// TIA Portal V20 export
FUNCTION_BLOCK "CentralShifter_SideShifters"   // FB17, LAD
{ S7_Optimized_Access := 'TRUE' }
// stored: MemoryReserve 100, SetENOAutomatically false
   VAR_INPUT
      In_Side_Drive_Pos : Bool;
      Position_CS : Int;
   END_VAR
   VAR_OUTPUT
      qLeftSide_in_Mid : Bool;
      qRightSide_in_Mid : Bool;
   END_VAR
   VAR
      Side_Hydraulic_CS_RL { S7_SetPoint := 'True'} : "Side_Hydraulic";
      Side_Hydraulic_CS_RR { S7_SetPoint := 'True'} : "Side_Hydraulic";
      Side_Driver_CS { S7_SetPoint := 'True'} : "Side_Driver";
      RL_Speed { S7_SetPoint := 'True'} : Int;
      RP_Speed : Int;
      CentralShifter_Side_Auto_Instance { S7_SetPoint := 'True'} : "CentralShifter_Side_Auto";
      SL_Auto_Speed { S7_SetPoint := 'True'} : Int;
      SR_Auto_Speed : Int;
      SL_Auto_Forward : Bool;
      SL_Auto_Backward : Bool;
      SR_Auto_Forward : Bool;
      SR_Auto_Backward : Bool;
      Sides_In_Position : Bool;
      Sides_In_H3_Pos : Bool;
      Sides_In_H5_Pos : Bool;
      Sides_In_CS_Pos : Bool;
      LightUp : Bool;
      LightMid : Bool;
      LightDown : Bool;
      SR_Error_Laser : Bool;
      SL_Error_Laser : Bool;
      Auto_Position_RL_Up : DInt;
      Auto_Position_RL_Mid : DInt;
      Auto_Position_RL_Down : DInt;
      Auto_Position_RR_Up : DInt;
      Auto_Position_RR_Mid : DInt;
      Auto_Position_RR_Down : DInt;
      Auto_Correction_RR : Int;
   END_VAR
   VAR RETAIN
      Stations : Array[7..13] of "CS_Sides_Stations";
   END_VAR
   VAR
      Status_Side_Go_H3 { S7_SetPoint := 'True'} : Int;
      Status_Side_Go_H5 : Int;
      Status_Side_Go_CS : Int;
      Auto_Hydraulic_Permission_H3 : Bool;
      Auto_Hydraulic_Permission_H5 : Bool;
      Auto_Hydraulic_Up_Timer { S7_SetPoint := 'True'} : TP_TIME;
      Auto_Hydraulic_Down_Timer { S7_SetPoint := 'True'} : TP_TIME;
      Station_H3_Empty : Bool;
      Station_H5_Empty : Bool;
      CS_R1_Sen_Up : Bool;
      CS_R1_Sen_Down : Bool;
      CS_R2_Sen_Up : Bool;
      CS_R2_Sen_Down : Bool;
      Auto_hyd_Up : Bool;
      Auto_hyd_Down : Bool;
      Hyd_Up_Status : Int;
      Hyd_Down_Status : Int;
      CS_RL_Error_Hyd : Bool;
      CS_RR_Error_Hyd : Bool;
      CS_Error_Hyd : Bool;
      CS_Error_Drive : Bool;
   END_VAR
   VAR CONSTANT
      Tolerance : Int := 60;
   END_VAR
   // Stations[7].RL_H3_Pos := 13516;
   // Stations[8].RL_H3_Pos := 13505;
   // Stations[9].RL_H3_Pos := 13520;
   // Stations[10].RL_H3_Pos := 13522;
   // Stations[11].RL_H3_Pos := 13526;
   // Stations[12].RL_H3_Pos := 13505;
   // Stations[13].RL_H3_Pos := 13500;
   // Stations[7].RR_H3_Pos := 13523;
   // Stations[8].RR_H3_Pos := 13495;
   // Stations[9].RR_H3_Pos := 13518;
   // Stations[10].RR_H3_Pos := 13527;
   // Stations[11].RR_H3_Pos := 13524;
   // Stations[12..13].RR_H3_Pos := 13525;
   // Stations[7].RL_Mid_Pos := 7915;
   // Stations[8].RL_Mid_Pos := 7910;
   // Stations[9].RL_Mid_Pos := 7933;
   // Stations[10].RL_Mid_Pos := 7928;
   // Stations[11].RL_Mid_Pos := 7937;
   // Stations[12].RL_Mid_Pos := 7932;
   // Stations[13].RL_Mid_Pos := 7916;
   // Stations[7].RR_Mid_Pos := 7925;
   // Stations[8].RR_Mid_Pos := 7895;
   // Stations[9].RR_Mid_Pos := 7922;
   // Stations[10].RR_Mid_Pos := 7935;
   // Stations[11].RR_Mid_Pos := 7926;
   // Stations[12].RR_Mid_Pos := 7932;
   // Stations[13].RR_Mid_Pos := 7939;
   // Stations[7].RL_H5_Pos := 1930;
   // Stations[8].RL_H5_Pos := 1917;
   // Stations[9].RL_H5_Pos := 1928;
   // Stations[10].RL_H5_Pos := 1929;
   // Stations[11].RL_H5_Pos := 1936;
   // Stations[12].RL_H5_Pos := 1924;
   // Stations[13].RL_H5_Pos := 1918;
   // Stations[7].RR_H5_Pos := 1929;
   // Stations[8].RR_H5_Pos := 1900;
   // Stations[9].RR_H5_Pos := 1921;
   // Stations[10].RR_H5_Pos := 1933;
   // Stations[11].RR_H5_Pos := 1928;
   // Stations[12].RR_H5_Pos := 1934;
   // Stations[13].RR_H5_Pos := 1915;
   // Stations[7].Correction := -20;
   // Stations[8].Correction := -15;
   // Stations[9].Correction := -5;
   // Stations[11].Correction := 0;
   // Stations[12].Correction := 10;
   // Stations[13].Correction := 15;
BEGIN

REGION Network 1: Hydraulic_RL
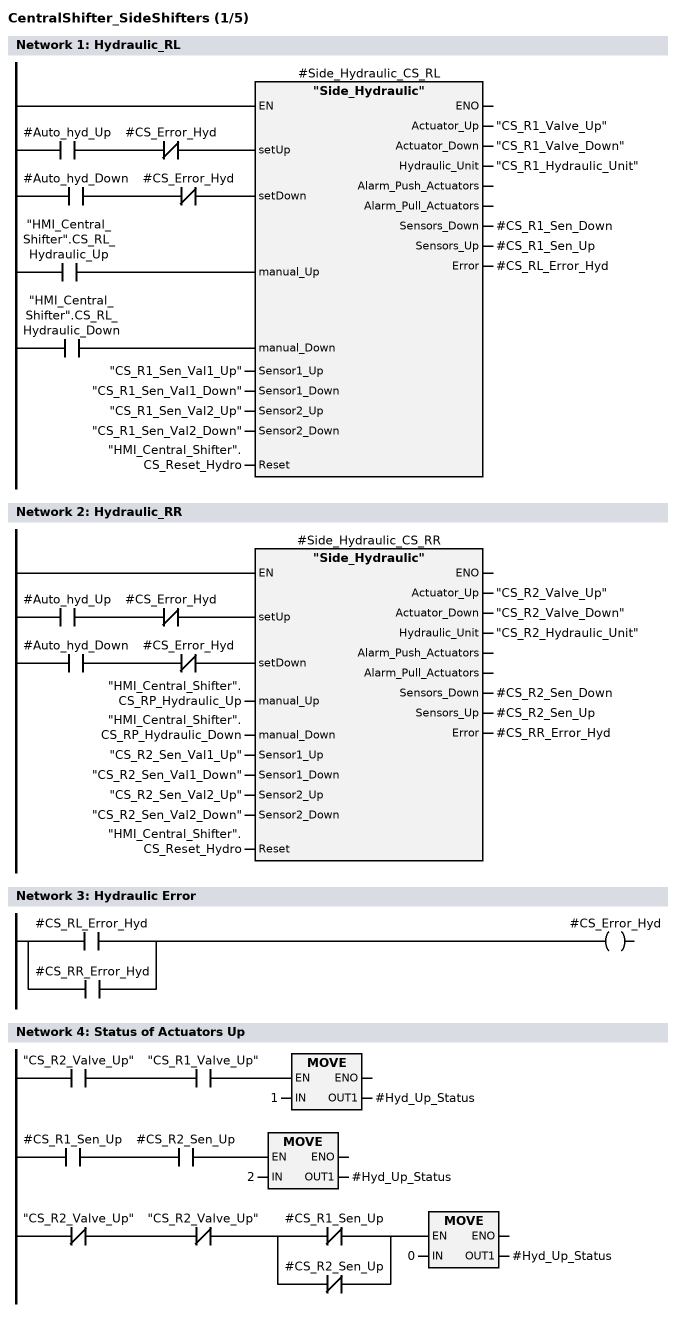
   RUNG wire#powerrail
      #Side_Hydraulic_CS_RL(setUp := wire#w1, setDown := wire#w2, manual_Up := wire#w3, manual_Down := wire#w4, Sensor1_Up := "CS_R1_Sen_Val1_Up", Sensor1_Down := "CS_R1_Sen_Val1_Down", Sensor2_Up := "CS_R1_Sen_Val2_Up", Sensor2_Down := "CS_R1_Sen_Val2_Down", Reset := "HMI_Central_Shifter".CS_Reset_Hydro, Actuator_Up => "CS_R1_Valve_Up", Actuator_Down => "CS_R1_Valve_Down", Hydraulic_Unit => "CS_R1_Hydraulic_Unit", Alarm_Push_Actuators =>, Alarm_Pull_Actuators =>, Sensors_Down => #CS_R1_Sen_Down, Sensors_Up => #CS_R1_Sen_Up, Error => #CS_RL_Error_Hyd)
   END_RUNG
   RUNG wire#powerrail
      Contact( #Auto_hyd_Up )
      I_Contact( #CS_Error_Hyd )
   END_RUNG wire#w1
   RUNG wire#powerrail
      Contact( #Auto_hyd_Down )
      I_Contact( #CS_Error_Hyd )
   END_RUNG wire#w2
   RUNG wire#powerrail
      Contact( "HMI_Central_Shifter".CS_RL_Hydraulic_Up )
   END_RUNG wire#w3
   RUNG wire#powerrail
      Contact( "HMI_Central_Shifter".CS_RL_Hydraulic_Down )
   END_RUNG wire#w4
   // the same network as SCL:
   #Side_Hydraulic_CS_RL(setUp := #Auto_hyd_Up AND NOT #CS_Error_Hyd,   // "Side_Hydraulic"
                         setDown := #Auto_hyd_Down AND NOT #CS_Error_Hyd,
                         manual_Up := "HMI_Central_Shifter".CS_RL_Hydraulic_Up,
                         manual_Down := "HMI_Central_Shifter".CS_RL_Hydraulic_Down,
                         Sensor1_Up := "CS_R1_Sen_Val1_Up",
                         Sensor1_Down := "CS_R1_Sen_Val1_Down",
                         Sensor2_Up := "CS_R1_Sen_Val2_Up",
                         Sensor2_Down := "CS_R1_Sen_Val2_Down",
                         Reset := "HMI_Central_Shifter".CS_Reset_Hydro,
                         Actuator_Up => "CS_R1_Valve_Up",
                         Actuator_Down => "CS_R1_Valve_Down",
                         Hydraulic_Unit => "CS_R1_Hydraulic_Unit",
                         Sensors_Down => #CS_R1_Sen_Down,
                         Sensors_Up => #CS_R1_Sen_Up,
                         Error => #CS_RL_Error_Hyd);
END_REGION

REGION Network 2: Hydraulic_RR
   RUNG wire#powerrail
      #Side_Hydraulic_CS_RR(setUp := wire#w1, setDown := wire#w2, manual_Up := "HMI_Central_Shifter".CS_RP_Hydraulic_Up, manual_Down := "HMI_Central_Shifter".CS_RP_Hydraulic_Down, Sensor1_Up := "CS_R2_Sen_Val1_Up", Sensor1_Down := "CS_R2_Sen_Val1_Down", Sensor2_Up := "CS_R2_Sen_Val2_Up", Sensor2_Down := "CS_R2_Sen_Val2_Down", Reset := "HMI_Central_Shifter".CS_Reset_Hydro, Actuator_Up => "CS_R2_Valve_Up", Actuator_Down => "CS_R2_Valve_Down", Hydraulic_Unit => "CS_R2_Hydraulic_Unit", Alarm_Push_Actuators =>, Alarm_Pull_Actuators =>, Sensors_Down => #CS_R2_Sen_Down, Sensors_Up => #CS_R2_Sen_Up, Error => #CS_RR_Error_Hyd)
   END_RUNG
   RUNG wire#powerrail
      Contact( #Auto_hyd_Up )
      I_Contact( #CS_Error_Hyd )
   END_RUNG wire#w1
   RUNG wire#powerrail
      Contact( #Auto_hyd_Down )
      I_Contact( #CS_Error_Hyd )
   END_RUNG wire#w2
   // the same network as SCL:
   #Side_Hydraulic_CS_RR(setUp := #Auto_hyd_Up AND NOT #CS_Error_Hyd,   // "Side_Hydraulic"
                         setDown := #Auto_hyd_Down AND NOT #CS_Error_Hyd,
                         manual_Up := "HMI_Central_Shifter".CS_RP_Hydraulic_Up,
                         manual_Down := "HMI_Central_Shifter".CS_RP_Hydraulic_Down,
                         Sensor1_Up := "CS_R2_Sen_Val1_Up",
                         Sensor1_Down := "CS_R2_Sen_Val1_Down",
                         Sensor2_Up := "CS_R2_Sen_Val2_Up",
                         Sensor2_Down := "CS_R2_Sen_Val2_Down",
                         Reset := "HMI_Central_Shifter".CS_Reset_Hydro,
                         Actuator_Up => "CS_R2_Valve_Up",
                         Actuator_Down => "CS_R2_Valve_Down",
                         Hydraulic_Unit => "CS_R2_Hydraulic_Unit",
                         Sensors_Down => #CS_R2_Sen_Down,
                         Sensors_Up => #CS_R2_Sen_Up,
                         Error => #CS_RR_Error_Hyd);
END_REGION

REGION Network 3: Hydraulic Error
   RUNG wire#powerrail
      Contact( #CS_RL_Error_Hyd )
      wire#w1
      Coil( #CS_Error_Hyd )
   END_RUNG
   RUNG wire#powerrail
      Contact( #CS_RR_Error_Hyd )
   END_RUNG wire#w1
   // the same network as SCL:
   #CS_Error_Hyd := #CS_RL_Error_Hyd OR #CS_RR_Error_Hyd;
END_REGION

REGION Network 4: Status of Actuators Up
   RUNG wire#powerrail
      Contact( "CS_R2_Valve_Up" )
      Contact( "CS_R1_Valve_Up" )
      Move(in := 1, out1 => #Hyd_Up_Status)
   END_RUNG
   RUNG wire#powerrail
      Contact( #CS_R1_Sen_Up )
      Contact( #CS_R2_Sen_Up )
      Move(in := 2, out1 => #Hyd_Up_Status)
   END_RUNG
   RUNG wire#powerrail
      I_Contact( "CS_R2_Valve_Up" )
      I_Contact( "CS_R2_Valve_Up" )
      wire#w1
      I_Contact( #CS_R1_Sen_Up )
      wire#w2
      Move(in := 0, out1 => #Hyd_Up_Status)
   END_RUNG
   RUNG wire#w1
      I_Contact( #CS_R2_Sen_Up )
   END_RUNG wire#w2
   // the same network as SCL:
   IF "CS_R2_Valve_Up" AND "CS_R1_Valve_Up" THEN #Hyd_Up_Status := 1; END_IF;
   IF #CS_R1_Sen_Up AND #CS_R2_Sen_Up THEN #Hyd_Up_Status := 2; END_IF;
   IF NOT "CS_R2_Valve_Up" AND NOT "CS_R2_Valve_Up" AND (NOT #CS_R1_Sen_Up OR NOT #CS_R2_Sen_Up) THEN
       #Hyd_Up_Status := 0;
   END_IF;
END_REGION

REGION Network 5: Status of Actuators Down
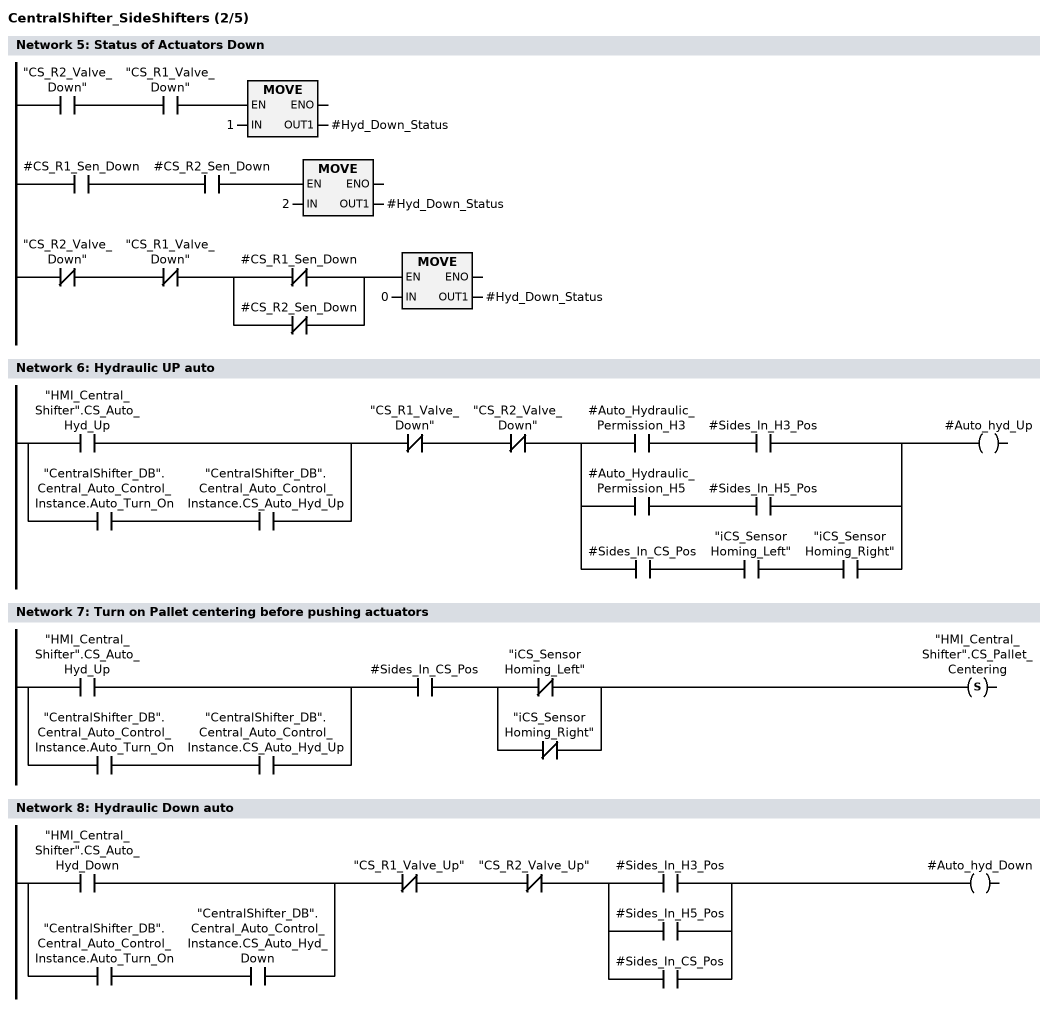
   RUNG wire#powerrail
      Contact( "CS_R2_Valve_Down" )
      Contact( "CS_R1_Valve_Down" )
      Move(in := 1, out1 => #Hyd_Down_Status)
   END_RUNG
   RUNG wire#powerrail
      Contact( #CS_R1_Sen_Down )
      Contact( #CS_R2_Sen_Down )
      Move(in := 2, out1 => #Hyd_Down_Status)
   END_RUNG
   RUNG wire#powerrail
      I_Contact( "CS_R2_Valve_Down" )
      I_Contact( "CS_R1_Valve_Down" )
      wire#w1
      I_Contact( #CS_R1_Sen_Down )
      wire#w2
      Move(in := 0, out1 => #Hyd_Down_Status)
   END_RUNG
   RUNG wire#w1
      I_Contact( #CS_R2_Sen_Down )
   END_RUNG wire#w2
   // the same network as SCL:
   IF "CS_R2_Valve_Down" AND "CS_R1_Valve_Down" THEN #Hyd_Down_Status := 1; END_IF;
   IF #CS_R1_Sen_Down AND #CS_R2_Sen_Down THEN #Hyd_Down_Status := 2; END_IF;
   IF NOT "CS_R2_Valve_Down" AND NOT "CS_R1_Valve_Down" AND (NOT #CS_R1_Sen_Down OR NOT #CS_R2_Sen_Down) THEN
       #Hyd_Down_Status := 0;
   END_IF;
END_REGION

REGION Network 6: Hydraulic UP auto
   RUNG wire#powerrail
      Contact( "HMI_Central_Shifter".CS_Auto_Hyd_Up )
      wire#w1
      I_Contact( "CS_R1_Valve_Down" )
      I_Contact( "CS_R2_Valve_Down" )
      wire#w2
      Contact( #Auto_Hydraulic_Permission_H3 )
      Contact( #Sides_In_H3_Pos )
      wire#w3
      Coil( #Auto_hyd_Up )
   END_RUNG
   RUNG wire#powerrail
      Contact( "CentralShifter_DB".Central_Auto_Control_Instance.Auto_Turn_On )
      Contact( "CentralShifter_DB".Central_Auto_Control_Instance.CS_Auto_Hyd_Up )
   END_RUNG wire#w1
   RUNG wire#w2
      Contact( #Auto_Hydraulic_Permission_H5 )
      Contact( #Sides_In_H5_Pos )
   END_RUNG wire#w3
   RUNG wire#w2
      Contact( #Sides_In_CS_Pos )
      Contact( "iCS_SensorHoming_Left" )
      Contact( "iCS_SensorHoming_Right" )
   END_RUNG wire#w3
   // the same network as SCL:
   #Auto_hyd_Up := ("HMI_Central_Shifter".CS_Auto_Hyd_Up OR ("CentralShifter_DB".Central_Auto_Control_Instance.Auto_Turn_On AND "CentralShifter_DB".Central_Auto_Control_Instance.CS_Auto_Hyd_Up)) AND NOT "CS_R1_Valve_Down" AND NOT "CS_R2_Valve_Down" AND ((#Auto_Hydraulic_Permission_H3 AND #Sides_In_H3_Pos) OR (#Auto_Hydraulic_Permission_H5 AND #Sides_In_H5_Pos) OR (#Sides_In_CS_Pos AND "iCS_SensorHoming_Left" AND "iCS_SensorHoming_Right"));
END_REGION

REGION Network 7: Turn on Pallet centering before pushing actuators
   RUNG wire#powerrail
      Contact( "HMI_Central_Shifter".CS_Auto_Hyd_Up )
      wire#w1
      Contact( #Sides_In_CS_Pos )
      wire#w2
      I_Contact( "iCS_SensorHoming_Left" )
      wire#w3
      S_Coil( "HMI_Central_Shifter".CS_Pallet_Centering )
   END_RUNG
   RUNG wire#powerrail
      Contact( "CentralShifter_DB".Central_Auto_Control_Instance.Auto_Turn_On )
      Contact( "CentralShifter_DB".Central_Auto_Control_Instance.CS_Auto_Hyd_Up )
   END_RUNG wire#w1
   RUNG wire#w2
      I_Contact( "iCS_SensorHoming_Right" )
   END_RUNG wire#w3
   // the same network as SCL:
   IF ("HMI_Central_Shifter".CS_Auto_Hyd_Up OR ("CentralShifter_DB".Central_Auto_Control_Instance.Auto_Turn_On AND "CentralShifter_DB".Central_Auto_Control_Instance.CS_Auto_Hyd_Up)) AND #Sides_In_CS_Pos AND (NOT "iCS_SensorHoming_Left" OR NOT "iCS_SensorHoming_Right") THEN
       "HMI_Central_Shifter".CS_Pallet_Centering := TRUE;
   END_IF;
END_REGION

REGION Network 8: Hydraulic Down auto
   RUNG wire#powerrail
      Contact( "HMI_Central_Shifter".CS_Auto_Hyd_Down )
      wire#w1
      I_Contact( "CS_R1_Valve_Up" )
      I_Contact( "CS_R2_Valve_Up" )
      wire#w2
      Contact( #Sides_In_H3_Pos )
      wire#w3
      Coil( #Auto_hyd_Down )
   END_RUNG
   RUNG wire#powerrail
      Contact( "CentralShifter_DB".Central_Auto_Control_Instance.Auto_Turn_On )
      Contact( "CentralShifter_DB".Central_Auto_Control_Instance.CS_Auto_Hyd_Down )
   END_RUNG wire#w1
   RUNG wire#w2
      Contact( #Sides_In_H5_Pos )
   END_RUNG wire#w3
   RUNG wire#w2
      Contact( #Sides_In_CS_Pos )
   END_RUNG wire#w3
   // the same network as SCL:
   #Auto_hyd_Down := ("HMI_Central_Shifter".CS_Auto_Hyd_Down OR ("CentralShifter_DB".Central_Auto_Control_Instance.Auto_Turn_On AND "CentralShifter_DB".Central_Auto_Control_Instance.CS_Auto_Hyd_Down)) AND NOT "CS_R1_Valve_Up" AND NOT "CS_R2_Valve_Up" AND (#Sides_In_H3_Pos OR #Sides_In_H5_Pos OR #Sides_In_CS_Pos);
END_REGION

REGION Network 9: Laser Error
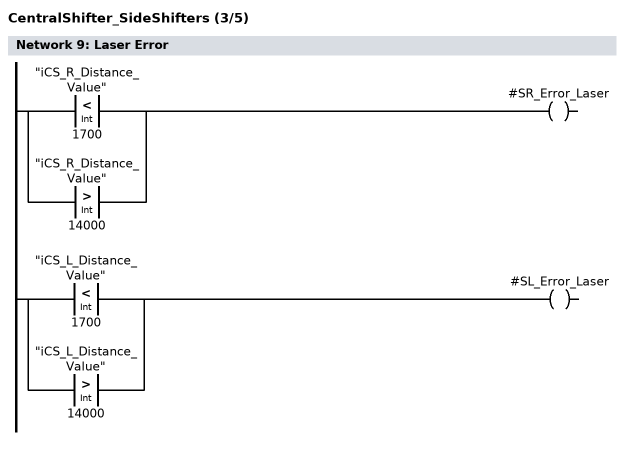
   RUNG wire#powerrail
      { S7_Templates := "SrcType := Int" } LT_Contact(in1 := "iCS_R_Distance_Value", in2 := 1700)
      wire#w1
      Coil( #SR_Error_Laser )
   END_RUNG
   RUNG wire#powerrail
      { S7_Templates := "SrcType := Int" } GT_Contact(in1 := "iCS_R_Distance_Value", in2 := 14000)
   END_RUNG wire#w1
   RUNG wire#powerrail
      { S7_Templates := "SrcType := Int" } LT_Contact(in1 := "iCS_L_Distance_Value", in2 := 1700)
      wire#w2
      Coil( #SL_Error_Laser )
   END_RUNG
   RUNG wire#powerrail
      { S7_Templates := "SrcType := Int" } GT_Contact(in1 := "iCS_L_Distance_Value", in2 := 14000)
   END_RUNG wire#w2
   // the same network as SCL:
   #SR_Error_Laser := ("iCS_R_Distance_Value" < 1700) OR ("iCS_R_Distance_Value" > 14000);
   #SL_Error_Laser := ("iCS_L_Distance_Value" < 1700) OR ("iCS_L_Distance_Value" > 14000);
END_REGION

REGION Network 10 (SCL): Setting SIDE positions by CS_POS
   CASE #Position_CS OF
       7..13:
           #Auto_Position_RL_Up := #Stations[#Position_CS].RL_H3_Pos;
           #Auto_Position_RR_Up := #Stations[#Position_CS].RR_H3_Pos;
           #Auto_Position_RL_Mid := #Stations[#Position_CS].RL_Mid_Pos;
           #Auto_Position_RR_Mid := #Stations[#Position_CS].RR_Mid_Pos;
           #Auto_Position_RL_Down := #Stations[#Position_CS].RL_H5_Pos;
           #Auto_Position_RR_Down := #Stations[#Position_CS].RR_H5_Pos;
           #Auto_Correction_RR := #Stations[#Position_CS].Correction;
       ELSE

           #Auto_Position_RL_Up := 0;
           #Auto_Position_RR_Up := 0;
           #Auto_Position_RL_Mid := 0;
           #Auto_Position_RR_Mid := 0;
           #Auto_Position_RL_Down := 0;
           #Auto_Position_RR_Down := 0;
           #Auto_Correction_RR := 0;
   END_CASE;
END_REGION

REGION Network 11 (SCL): Perform centering during hyd up
   CASE #Position_CS OF
       7..13:
           IF #Sides_In_H3_Pos AND ("HMI_Central_Shifter".CS_Auto_Hyd_Up OR ("CentralShifter_DB".Central_Auto_Control_Instance.Auto_Turn_On AND "CentralShifter_DB".Central_Auto_Control_Instance.CS_Auto_Hyd_Up)) AND NOT "System_To_Moving_Pallets_DB".Centering_Status[#Position_CS, 1] THEN
               "System_To_Moving_Pallets_DB".Centering_Perform[#Position_CS, 1] := 1;
           ELSIF #Sides_In_H5_Pos AND ("HMI_Central_Shifter".CS_Auto_Hyd_Up OR ("CentralShifter_DB".Central_Auto_Control_Instance.Auto_Turn_On AND "CentralShifter_DB".Central_Auto_Control_Instance.CS_Auto_Hyd_Up)) AND NOT "System_To_Moving_Pallets_DB".Centering_Status[#Position_CS, 3] THEN
               "System_To_Moving_Pallets_DB".Centering_Perform[#Position_CS, 3] := 1;
           END_IF;
   END_CASE;
END_REGION

REGION Network 12 (SCL): Permission to hyd up auto
   CASE #Position_CS OF
       7..13:
           IF "System_To_Moving_Pallets_DB".Centering_Status[#Position_CS, 1] THEN

               #Auto_Hydraulic_Permission_H3 := 1;
           ELSE
               #Auto_Hydraulic_Permission_H3 := 0;
           END_IF;

           IF "System_To_Moving_Pallets_DB".Centering_Status[#Position_CS, 3] THEN

               #Auto_Hydraulic_Permission_H5 := 1;
           ELSE
               #Auto_Hydraulic_Permission_H5 := 0;
           END_IF;

   END_CASE;
END_REGION

REGION Network 13 (SCL): Stations empty
   CASE #Position_CS OF
       7..13:
               #Station_H3_Empty := "Pallets_Stations".Stations[4, #Position_CS-3].IsEmpty;

               #Station_H5_Empty := "Pallets_Stations".Stations[2, #Position_CS-2].IsEmpty;

   END_CASE;
END_REGION

REGION Network 14: SIde Drivers
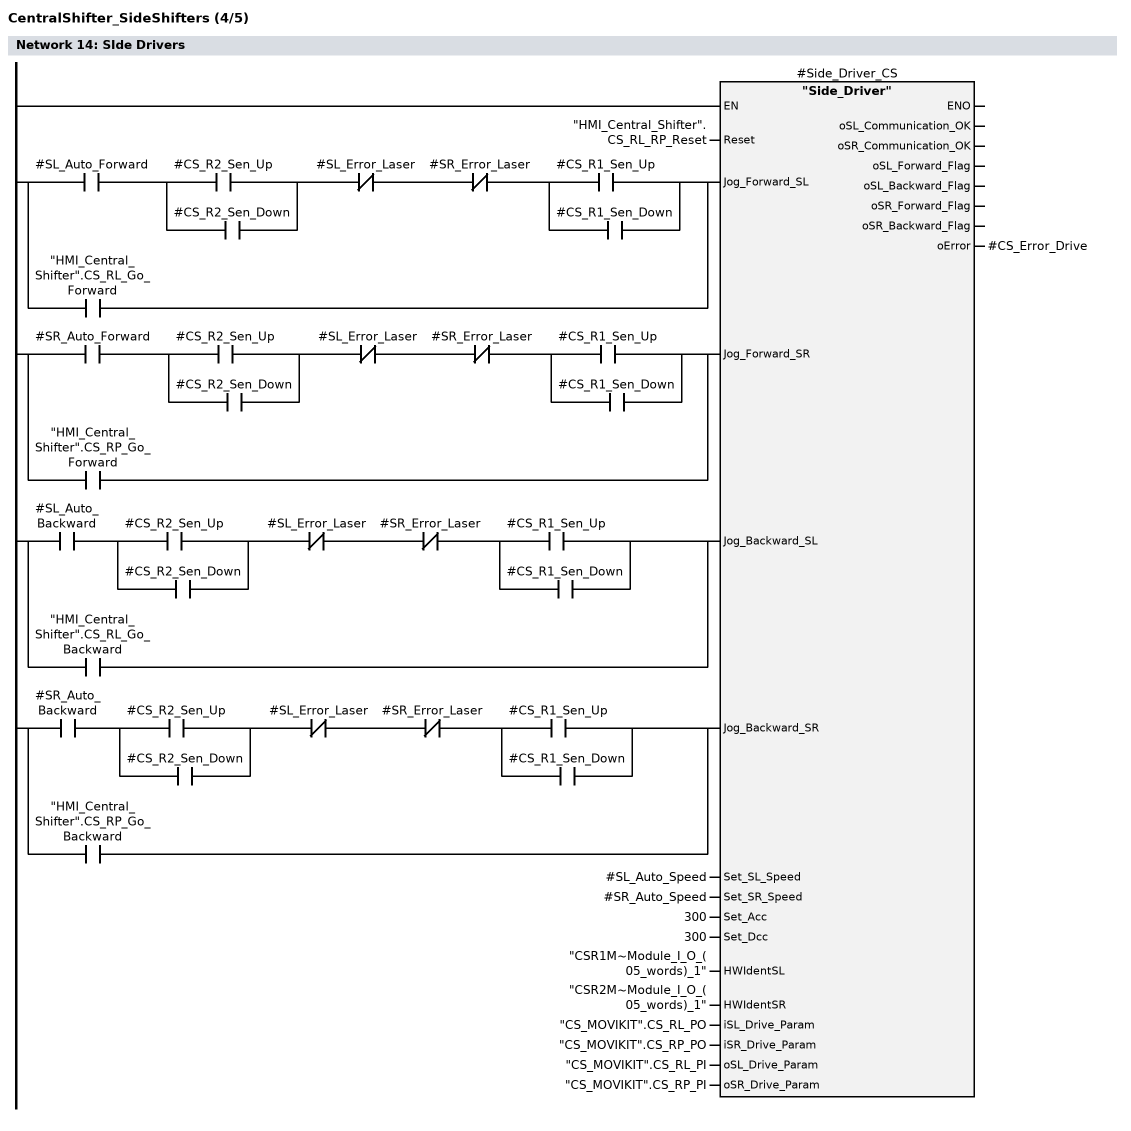
   RUNG wire#powerrail
      #Side_Driver_CS(Jog_Forward_SL := wire#w4, Jog_Forward_SR := wire#w8, Jog_Backward_SL := wire#w12, Jog_Backward_SR := wire#w16, Reset := "HMI_Central_Shifter".CS_RL_RP_Reset, Set_SL_Speed := #SL_Auto_Speed, Set_SR_Speed := #SR_Auto_Speed, Set_Acc := 300, Set_Dcc := 300, HWIdentSL := "CSR1M~Module_I_O_(05_words)_1", HWIdentSR := "CSR2M~Module_I_O_(05_words)_1", iSL_Drive_Param := "CS_MOVIKIT".CS_RL_PO, iSR_Drive_Param := "CS_MOVIKIT".CS_RP_PO, oSL_Drive_Param := "CS_MOVIKIT".CS_RL_PI, oSR_Drive_Param := "CS_MOVIKIT".CS_RP_PI, oSL_Communication_OK =>, oSR_Communication_OK =>, oSL_Forward_Flag =>, oSL_Backward_Flag =>, oSR_Forward_Flag =>, oSR_Backward_Flag =>, oError => #CS_Error_Drive)
   END_RUNG
   RUNG wire#powerrail
      Contact( #SL_Auto_Forward )
      wire#w1
      Contact( #CS_R2_Sen_Up )
      wire#w2
      I_Contact( #SL_Error_Laser )
      I_Contact( #SR_Error_Laser )
      wire#w3
      Contact( #CS_R1_Sen_Up )
   END_RUNG wire#w4
   RUNG wire#w1
      Contact( #CS_R2_Sen_Down )
   END_RUNG wire#w2
   RUNG wire#w3
      Contact( #CS_R1_Sen_Down )
   END_RUNG wire#w4
   RUNG wire#powerrail
      Contact( "HMI_Central_Shifter".CS_RL_Go_Forward )
   END_RUNG wire#w4
   RUNG wire#powerrail
      Contact( #SR_Auto_Forward )
      wire#w5
      Contact( #CS_R2_Sen_Up )
      wire#w6
      I_Contact( #SL_Error_Laser )
      I_Contact( #SR_Error_Laser )
      wire#w7
      Contact( #CS_R1_Sen_Up )
   END_RUNG wire#w8
   RUNG wire#w5
      Contact( #CS_R2_Sen_Down )
   END_RUNG wire#w6
   RUNG wire#w7
      Contact( #CS_R1_Sen_Down )
   END_RUNG wire#w8
   RUNG wire#powerrail
      Contact( "HMI_Central_Shifter".CS_RP_Go_Forward )
   END_RUNG wire#w8
   RUNG wire#powerrail
      Contact( #SL_Auto_Backward )
      wire#w9
      Contact( #CS_R2_Sen_Up )
      wire#w10
      I_Contact( #SL_Error_Laser )
      I_Contact( #SR_Error_Laser )
      wire#w11
      Contact( #CS_R1_Sen_Up )
   END_RUNG wire#w12
   RUNG wire#w9
      Contact( #CS_R2_Sen_Down )
   END_RUNG wire#w10
   RUNG wire#w11
      Contact( #CS_R1_Sen_Down )
   END_RUNG wire#w12
   RUNG wire#powerrail
      Contact( "HMI_Central_Shifter".CS_RL_Go_Backward )
   END_RUNG wire#w12
   RUNG wire#powerrail
      Contact( #SR_Auto_Backward )
      wire#w13
      Contact( #CS_R2_Sen_Up )
      wire#w14
      I_Contact( #SL_Error_Laser )
      I_Contact( #SR_Error_Laser )
      wire#w15
      Contact( #CS_R1_Sen_Up )
   END_RUNG wire#w16
   RUNG wire#w13
      Contact( #CS_R2_Sen_Down )
   END_RUNG wire#w14
   RUNG wire#w15
      Contact( #CS_R1_Sen_Down )
   END_RUNG wire#w16
   RUNG wire#powerrail
      Contact( "HMI_Central_Shifter".CS_RP_Go_Backward )
   END_RUNG wire#w16
   // the same network as SCL:
   #Side_Driver_CS(Reset := "HMI_Central_Shifter".CS_RL_RP_Reset,   // "Side_Driver"
                   Jog_Forward_SL := (#SL_Auto_Forward AND (#CS_R2_Sen_Up OR #CS_R2_Sen_Down) AND NOT #SL_Error_Laser AND NOT #SR_Error_Laser AND (#CS_R1_Sen_Up OR #CS_R1_Sen_Down)) OR "HMI_Central_Shifter".CS_RL_Go_Forward,
                   Jog_Forward_SR := (#SR_Auto_Forward AND (#CS_R2_Sen_Up OR #CS_R2_Sen_Down) AND NOT #SL_Error_Laser AND NOT #SR_Error_Laser AND (#CS_R1_Sen_Up OR #CS_R1_Sen_Down)) OR "HMI_Central_Shifter".CS_RP_Go_Forward,
                   Jog_Backward_SL := (#SL_Auto_Backward AND (#CS_R2_Sen_Up OR #CS_R2_Sen_Down) AND NOT #SL_Error_Laser AND NOT #SR_Error_Laser AND (#CS_R1_Sen_Up OR #CS_R1_Sen_Down)) OR "HMI_Central_Shifter".CS_RL_Go_Backward,
                   Jog_Backward_SR := (#SR_Auto_Backward AND (#CS_R2_Sen_Up OR #CS_R2_Sen_Down) AND NOT #SL_Error_Laser AND NOT #SR_Error_Laser AND (#CS_R1_Sen_Up OR #CS_R1_Sen_Down)) OR "HMI_Central_Shifter".CS_RP_Go_Backward,
                   Set_SL_Speed := #SL_Auto_Speed,
                   Set_SR_Speed := #SR_Auto_Speed,
                   Set_Acc := 300,
                   Set_Dcc := 300,
                   HWIdentSL := "CSR1M~Module_I_O_(05_words)_1",
                   HWIdentSR := "CSR2M~Module_I_O_(05_words)_1",
                   iSL_Drive_Param := "CS_MOVIKIT".CS_RL_PO,
                   iSR_Drive_Param := "CS_MOVIKIT".CS_RP_PO,
                   oSL_Drive_Param := "CS_MOVIKIT".CS_RL_PI,
                   oSR_Drive_Param := "CS_MOVIKIT".CS_RP_PI,
                   oError => #CS_Error_Drive);
END_REGION

REGION Network 15 (SCL): Limit positions of Sides
   IF #Auto_Position_RL_Down > 14000 THEN
       #Auto_Position_RL_Down := 14000;
   ELSIF #Auto_Position_RL_Down < 1800 THEN
       #Auto_Position_RL_Down := 1800;
   END_IF;

   IF #Auto_Position_RL_Up > 14000 THEN
       #Auto_Position_RL_Up := 14000;
   ELSIF #Auto_Position_RL_Up < 1800 THEN
       #Auto_Position_RL_Up := 1800;
   END_IF;

   IF #Auto_Position_RR_Down > 14000 THEN
       #Auto_Position_RR_Down := 14000;
   ELSIF #Auto_Position_RR_Down < 1800 THEN
       #Auto_Position_RR_Down := 1800;
   END_IF;

   IF #Auto_Position_RR_Up > 14000 THEN
       #Auto_Position_RR_Up := 14000;
   ELSIF #Auto_Position_RR_Up < 1800 THEN
       #Auto_Position_RR_Up := 1800;
   END_IF;
END_REGION

REGION Network 16: CS Side Auto
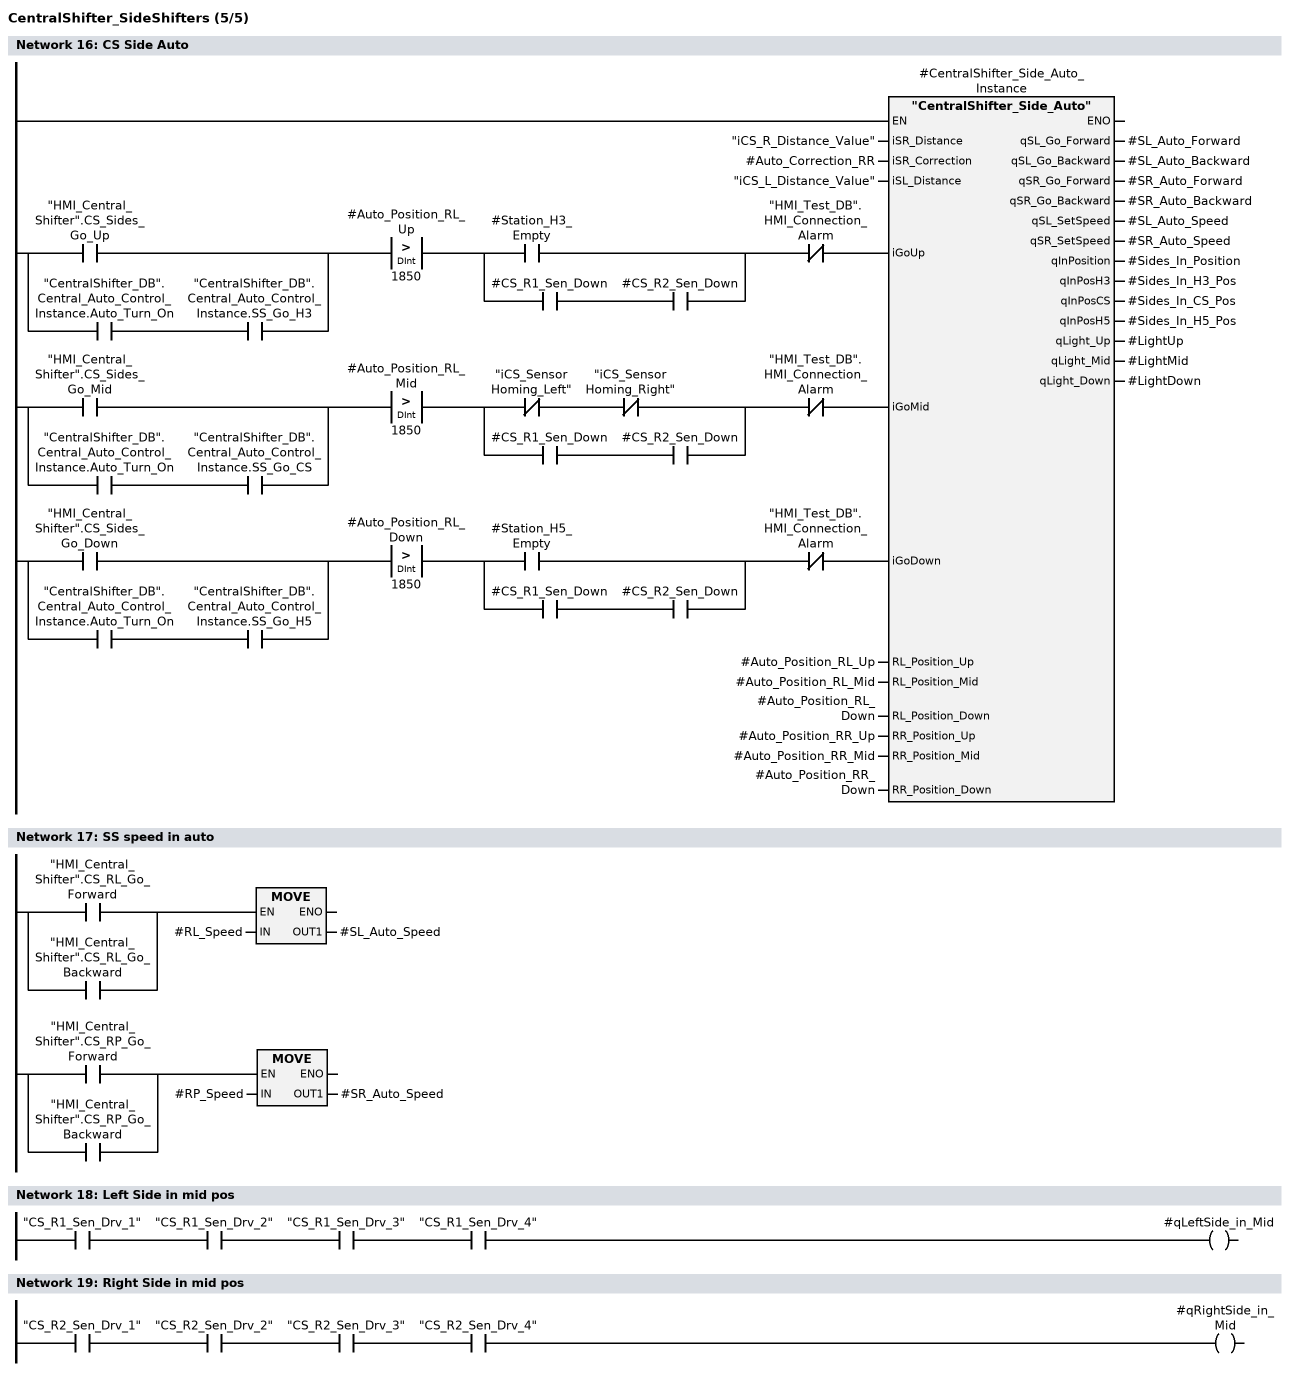
   RUNG wire#powerrail
      #CentralShifter_Side_Auto_Instance(iGoUp := wire#w4, iGoMid := wire#w8, iGoDown := wire#w12, iSR_Distance := "iCS_R_Distance_Value", iSR_Correction := #Auto_Correction_RR, iSL_Distance := "iCS_L_Distance_Value", RL_Position_Up := #Auto_Position_RL_Up, RL_Position_Mid := #Auto_Position_RL_Mid, RL_Position_Down := #Auto_Position_RL_Down, RR_Position_Up := #Auto_Position_RR_Up, RR_Position_Mid := #Auto_Position_RR_Mid, RR_Position_Down := #Auto_Position_RR_Down, qSL_Go_Forward => #SL_Auto_Forward, qSL_Go_Backward => #SL_Auto_Backward, qSR_Go_Forward => #SR_Auto_Forward, qSR_Go_Backward => #SR_Auto_Backward, qSL_SetSpeed => #SL_Auto_Speed, qSR_SetSpeed => #SR_Auto_Speed, qInPosition => #Sides_In_Position, qInPosH3 => #Sides_In_H3_Pos, qInPosCS => #Sides_In_CS_Pos, qInPosH5 => #Sides_In_H5_Pos, qLight_Up => #LightUp, qLight_Mid => #LightMid, qLight_Down => #LightDown)
   END_RUNG
   RUNG wire#powerrail
      Contact( "HMI_Central_Shifter".CS_Sides_Go_Up )
      wire#w1
      { S7_Templates := "SrcType := DInt" } GT_Contact(in1 := #Auto_Position_RL_Up, in2 := 1850)
      wire#w2
      Contact( #Station_H3_Empty )
      wire#w3
      I_Contact( "HMI_Test_DB".HMI_Connection_Alarm )
   END_RUNG wire#w4
   RUNG wire#powerrail
      Contact( "CentralShifter_DB".Central_Auto_Control_Instance.Auto_Turn_On )
      Contact( "CentralShifter_DB".Central_Auto_Control_Instance.SS_Go_H3 )
   END_RUNG wire#w1
   RUNG wire#w2
      Contact( #CS_R1_Sen_Down )
      Contact( #CS_R2_Sen_Down )
   END_RUNG wire#w3
   RUNG wire#powerrail
      Contact( "HMI_Central_Shifter".CS_Sides_Go_Mid )
      wire#w5
      { S7_Templates := "SrcType := DInt" } GT_Contact(in1 := #Auto_Position_RL_Mid, in2 := 1850)
      wire#w6
      I_Contact( "iCS_SensorHoming_Left" )
      I_Contact( "iCS_SensorHoming_Right" )
      wire#w7
      I_Contact( "HMI_Test_DB".HMI_Connection_Alarm )
   END_RUNG wire#w8
   RUNG wire#powerrail
      Contact( "CentralShifter_DB".Central_Auto_Control_Instance.Auto_Turn_On )
      Contact( "CentralShifter_DB".Central_Auto_Control_Instance.SS_Go_CS )
   END_RUNG wire#w5
   RUNG wire#w6
      Contact( #CS_R1_Sen_Down )
      Contact( #CS_R2_Sen_Down )
   END_RUNG wire#w7
   RUNG wire#powerrail
      Contact( "HMI_Central_Shifter".CS_Sides_Go_Down )
      wire#w9
      { S7_Templates := "SrcType := DInt" } GT_Contact(in1 := #Auto_Position_RL_Down, in2 := 1850)
      wire#w10
      Contact( #Station_H5_Empty )
      wire#w11
      I_Contact( "HMI_Test_DB".HMI_Connection_Alarm )
   END_RUNG wire#w12
   RUNG wire#powerrail
      Contact( "CentralShifter_DB".Central_Auto_Control_Instance.Auto_Turn_On )
      Contact( "CentralShifter_DB".Central_Auto_Control_Instance.SS_Go_H5 )
   END_RUNG wire#w9
   RUNG wire#w10
      Contact( #CS_R1_Sen_Down )
      Contact( #CS_R2_Sen_Down )
   END_RUNG wire#w11
   // the same network as SCL:
   #CentralShifter_Side_Auto_Instance(iSR_Distance := "iCS_R_Distance_Value",   // "CentralShifter_Side_Auto"
                           iSR_Correction := #Auto_Correction_RR,
                           iSL_Distance := "iCS_L_Distance_Value",
                           iGoUp := ("HMI_Central_Shifter".CS_Sides_Go_Up OR ("CentralShifter_DB".Central_Auto_Control_Instance.Auto_Turn_On AND "CentralShifter_DB".Central_Auto_Control_Instance.SS_Go_H3)) AND (#Auto_Position_RL_Up > 1850) AND (#Station_H3_Empty OR (#CS_R1_Sen_Down AND #CS_R2_Sen_Down)) AND NOT "HMI_Test_DB".HMI_Connection_Alarm,
                           iGoMid := ("HMI_Central_Shifter".CS_Sides_Go_Mid OR ("CentralShifter_DB".Central_Auto_Control_Instance.Auto_Turn_On AND "CentralShifter_DB".Central_Auto_Control_Instance.SS_Go_CS)) AND (#Auto_Position_RL_Mid > 1850) AND ((NOT "iCS_SensorHoming_Left" AND NOT "iCS_SensorHoming_Right") OR (#CS_R1_Sen_Down AND #CS_R2_Sen_Down)) AND NOT "HMI_Test_DB".HMI_Connection_Alarm,
                           iGoDown := ("HMI_Central_Shifter".CS_Sides_Go_Down OR ("CentralShifter_DB".Central_Auto_Control_Instance.Auto_Turn_On AND "CentralShifter_DB".Central_Auto_Control_Instance.SS_Go_H5)) AND (#Auto_Position_RL_Down > 1850) AND (#Station_H5_Empty OR (#CS_R1_Sen_Down AND #CS_R2_Sen_Down)) AND NOT "HMI_Test_DB".HMI_Connection_Alarm,
                           RL_Position_Up := #Auto_Position_RL_Up,
                           RL_Position_Mid := #Auto_Position_RL_Mid,
                           RL_Position_Down := #Auto_Position_RL_Down,
                           RR_Position_Up := #Auto_Position_RR_Up,
                           RR_Position_Mid := #Auto_Position_RR_Mid,
                           RR_Position_Down := #Auto_Position_RR_Down,
                           qSL_Go_Forward => #SL_Auto_Forward,
                           qSL_Go_Backward => #SL_Auto_Backward,
                           qSR_Go_Forward => #SR_Auto_Forward,
                           qSR_Go_Backward => #SR_Auto_Backward,
                           qSL_SetSpeed => #SL_Auto_Speed,
                           qSR_SetSpeed => #SR_Auto_Speed,
                           qInPosition => #Sides_In_Position,
                           qInPosH3 => #Sides_In_H3_Pos,
                           qInPosCS => #Sides_In_CS_Pos,
                           qInPosH5 => #Sides_In_H5_Pos,
                           qLight_Up => #LightUp,
                           qLight_Mid => #LightMid,
                           qLight_Down => #LightDown);
END_REGION

REGION Network 17: SS speed in auto
   RUNG wire#powerrail
      Contact( "HMI_Central_Shifter".CS_RL_Go_Forward )
      wire#w1
      Move(in := #RL_Speed, out1 => #SL_Auto_Speed)
   END_RUNG
   RUNG wire#powerrail
      Contact( "HMI_Central_Shifter".CS_RL_Go_Backward )
   END_RUNG wire#w1
   RUNG wire#powerrail
      Contact( "HMI_Central_Shifter".CS_RP_Go_Forward )
      wire#w2
      Move(in := #RP_Speed, out1 => #SR_Auto_Speed)
   END_RUNG
   RUNG wire#powerrail
      Contact( "HMI_Central_Shifter".CS_RP_Go_Backward )
   END_RUNG wire#w2
   // the same network as SCL:
   IF "HMI_Central_Shifter".CS_RL_Go_Forward OR "HMI_Central_Shifter".CS_RL_Go_Backward THEN
       #SL_Auto_Speed := #RL_Speed;
   END_IF;
   IF "HMI_Central_Shifter".CS_RP_Go_Forward OR "HMI_Central_Shifter".CS_RP_Go_Backward THEN
       #SR_Auto_Speed := #RP_Speed;
   END_IF;
END_REGION

REGION Network 18: Left Side in mid pos
   RUNG wire#powerrail
      Contact( "CS_R1_Sen_Drv_1" )
      Contact( "CS_R1_Sen_Drv_2" )
      Contact( "CS_R1_Sen_Drv_3" )
      Contact( "CS_R1_Sen_Drv_4" )
      Coil( #qLeftSide_in_Mid )
   END_RUNG
   // the same network as SCL:
   #qLeftSide_in_Mid := "CS_R1_Sen_Drv_1" AND "CS_R1_Sen_Drv_2" AND "CS_R1_Sen_Drv_3" AND "CS_R1_Sen_Drv_4";
END_REGION

REGION Network 19: Right Side in mid pos
   RUNG wire#powerrail
      Contact( "CS_R2_Sen_Drv_1" )
      Contact( "CS_R2_Sen_Drv_2" )
      Contact( "CS_R2_Sen_Drv_3" )
      Contact( "CS_R2_Sen_Drv_4" )
      Coil( #qRightSide_in_Mid )
   END_RUNG
   // the same network as SCL:
   #qRightSide_in_Mid := "CS_R2_Sen_Drv_1" AND "CS_R2_Sen_Drv_2" AND "CS_R2_Sen_Drv_3" AND "CS_R2_Sen_Drv_4";
END_REGION

REGION Network 20 (SCL): Status - go to destinations
           IF "HMI_Central_Shifter".CS_Sides_Go_Up AND NOT #Sides_In_H3_Pos AND #In_Side_Drive_Pos THEN
               #Status_Side_Go_H3 := 1;
           ELSIF #Sides_In_H3_Pos THEN
               #Status_Side_Go_H3 := 2;
           ELSE
               #Status_Side_Go_H3 := 0;
           END_IF;

           IF "HMI_Central_Shifter".CS_Sides_Go_Down AND NOT #Sides_In_H5_Pos AND #In_Side_Drive_Pos THEN
               #Status_Side_Go_H5 := 1;
           ELSIF #Sides_In_H5_Pos THEN
               #Status_Side_Go_H5 := 2;
           ELSE
               #Status_Side_Go_H5 := 0;
           END_IF;

           IF "HMI_Central_Shifter".CS_Sides_Go_Mid AND NOT #Sides_In_CS_Pos AND #In_Side_Drive_Pos THEN
               #Status_Side_Go_CS := 1;
           ELSIF #Sides_In_CS_Pos THEN
               #Status_Side_Go_CS := 2;
           ELSE
               #Status_Side_Go_CS := 0;
           END_IF;
END_REGION
END_FUNCTION_BLOCK
